// TwinCAT 3 PLC project Lab2_2
// ProgramVersion: 3.1.4023.0
// libraries:
//   Tc2_Standard, * (Beckhoff Automation GmbH)
//   Tc2_System, * (Beckhoff Automation GmbH)
//   Tc3_Module, * (Beckhoff Automation GmbH)
// project tree:
//   / PlcTask.TcTTO
//   POUs/ MAIN.TcPOU
//   Task1/D_Task1/ E_SensorBrand.TcDUT
//   Task1/G_Task1/ GVL.TcGVL
//   Task1/P_Task1/ P_Prog1.TcPOU
//   Task2/D_Task2/ ST_Motor.TcDUT, ST_Timer.TcDUT
//   Task2/G_Task2/ G_Task2.TcGVL
//   Task2/P_Task2/ Deg_To_Rad.TcPOU, P_Task2.TcPOU, Updete_Motor_Parameters.TcPOU, Updete_Motor_Parameters_Reference.TcPOU
// real-time tasks:
//   TASK PlcTask: cycle T#10ms, priority 20, ADS port 350

CONFIGURATION Lab2_2
    RESOURCE PLC ON TwinCAT3
        TASK PlcTask(INTERVAL := T#10ms, PRIORITY := 20);
        PROGRAM MAIN WITH PlcTask : MAIN;
    END_RESOURCE
END_CONFIGURATION

// ---- Task1/D_Task1/E_SensorBrand.TcDUT
{attribute 'qualified_only'}
{attribute 'strict'}
TYPE E_SensorBrand :
(
	Sick,
	Pilz,
	Parker,
	Bosch
);
END_TYPE

// ---- Task2/D_Task2/ST_Motor.TcDUT
TYPE ST_Motor :
STRUCT
	fSpeedMax : REAL;
	fSpeedMin : REAL;
END_STRUCT
END_TYPE

// ---- Task2/D_Task2/ST_Timer.TcDUT
TYPE ST_Timer :
STRUCT
	bTimerStat : BOOL;
	bTimerOut : BOOL;
	tTimeElapsed : TIME;
	tTimer : TIME;
END_STRUCT
END_TYPE

// ---- Task1/G_Task1/GVL.TcGVL
{attribute 'qualified_only'}
VAR_GLOBAL
	dtCurrentdate : DATE_AND_TIME := DT#2023-02-13-19:58:39;
	tTimeVar : TIME := T#4S;
	aDateArray : ARRAY[0..3] OF DATE := [D#2023-02-07, D#2023-02-08, D#2023-02-09, D#2023-02-10];
	eSensor1 : E_SensorBrand := E_SensorBrand.Parker;
	bTimeStarter : BOOL := FALSE;
	bOutQ : BOOL;
	tElapseTime : TIME;
	fbTimer : TON := (PT := T#10S);
END_VAR

// ---- Task2/G_Task2/G_Task2.TcGVL
{attribute 'qualified_only'}
VAR_GLOBAL
	stTimer2 : ST_Timer := (tTimer := T#5S);
	fMotor1Rad : REAL;
	fMotor1Deg : REAL := 180;
	st_MotorParameters1 : ST_Motor;
	st_MotorParameters2 : ST_Motor;
END_VAR

// ---- POUs/MAIN.TcPOU
PROGRAM MAIN
VAR
END_VAR

P_Task2();

END_PROGRAM

// ---- Task2/P_Task2/P_Task2.TcPOU
PROGRAM P_Task2
VAR
	fbTof : TOF;
	fbRTrig : R_TRIG;
	bMotorUpdate : BOOL;
	fNewValue : REAL;
END_VAR

fbTof(IN := G_Task2.stTimer2.bTimerStat,
		PT := G_Task2.stTimer2.tTimer,
		Q => G_Task2.stTimer2.bTimerOut,
		ET => G_Task2.stTimer2.tTimeElapsed);
		
G_Task2.fMotor1Rad := Deg_To_Rad(fDeg := G_Task2.fMotor1Deg);

fbRTrig(CLK := bMotorUpdate);
Updete_Motor_Parameters(bUpdateValue := fbRTrig.Q, fNewValue := fNewValue, G_Task2.st_MotorParameters1);
Updete_Motor_Parameters_Reference(bUpdateValue := fbRTrig.Q, fNewValue := fNewValue, G_Task2.st_MotorParameters2);

END_PROGRAM

// ---- Task2/P_Task2/Deg_To_Rad.TcPOU
FUNCTION Deg_To_Rad : REAL
VAR_INPUT
	fDeg : REAL;
END_VAR
VAR
	fPi : REAL := 3.14159265359;
END_VAR

Deg_To_Rad := (fDeg * fPi)/180;

END_FUNCTION

// ---- Task2/P_Task2/Updete_Motor_Parameters.TcPOU
FUNCTION Updete_Motor_Parameters
VAR_INPUT
	bUpdateValue : BOOL;
	fNewValue : REAL;
	stMotorParameters : ST_Motor;
END_VAR
VAR
END_VAR

IF bUpdateValue = 1 THEN
	stMotorParameters.fSpeedMax := fNewValue;
ELSE
	stMotorParameters.fSpeedMax := stMotorParameters.fSpeedMax;
END_IF

END_FUNCTION

// ---- Task2/P_Task2/Updete_Motor_Parameters_Reference.TcPOU
FUNCTION Updete_Motor_Parameters_Reference
VAR_INPUT
	bUpdateValue : BOOL;
	fNewValue : REAL;
	stMotorParameters : REFERENCE TO ST_Motor;
END_VAR
VAR
END_VAR

IF bUpdateValue = 1 THEN
	stMotorParameters.fSpeedMax := fNewValue;
ELSE
	stMotorParameters.fSpeedMax := stMotorParameters.fSpeedMax;
END_IF

END_FUNCTION

// ---- Task1/P_Task1/P_Prog1.TcPOU
PROGRAM P_Prog1
VAR
	pDatePointer : POINTER TO DATE_AND_TIME := ADR(GVL.dtCurrentdate);
	nTimeRefrence : REFERENCE TO TIME := GVL.tTimeVar;
END_VAR

pDatePointer^ := DT#2023-02-08-15:31:19;
nTimeRefrence := T#2S;
GVL.aDateArray[2] := D#2023-02-25;
GVL.eSensor1 := E_SensorBrand.Bosch;
GVL.fbTimer(IN := GVL.bTimeStarter);
GVL.bOutQ := GVL.fbTimer.Q;
GVL.tElapseTime := GVL.fbTimer.ET;

END_PROGRAM
